(* CODESYS project mir3502tester_20200314.1.project

Project tree, tasks and I/O mapping:
  Device : Changsha Xiangji-ARM Cortex A9(xilinx zynq7000)-linux, Changsha Xiangji Hiden Technology Co.Ltd, version 3.5.10.40
    application Application
      libraries: Standard, * (System); SysFile, 3.5.15.0 (System); SysTypes2 Interfaces, * (System); SysShm, * (System); CAA Mathematics, * (CAA Technical Workgroup); CAA Net Base Services, * (CAA Technical Workgroup); SysTime, 3.5.9.0 (System); VisuDialogs, * (System); CAA Storage, 3.5.13.0 (CAA Technical Workgroup)
      task c_MainTask (cyclic, interval 20 ms, priority 20) calls prg_main
      task a_motion_tasks (cyclic, interval 10 ms, priority 5) calls EtherCAT_Master_SoftMotion.EtherCAT_Task
      program prg_main [ST]
    EtherCAT_Master_SoftMotion : EtherCAT Master SoftMotion, 3S - Smart Software Solutions GmbH, version 3.5.14.30
        settings: MasterCycleTime = 10000; MasterUseLRW = False; SlaveAutoRestart = True; NetworkName = 'eth0'; NetworkName = "eth0"; SelectNetworkByName = True; EnableTaskMessage = False; SrcAddress1 = 4784; SrcAddress2 = 3830812668
      MIR3502 : MIR3502, Cyber-MI, order no. MIR3502, version Revision=16#00000000
          settings: StationAlias = 0; DC sync0 cycletime = 10000; DC sync1 cycletime = 10000
          output Application.prg_main.mir3502_pwm01 : UINT  // PWM01-C35
          output Application.prg_main.mir3502_do00 : BIT  // DO00-C01
          input  Application.prg_main.mir3502_ai00 : UINT  // AI00-C20
          input  Application.prg_main.mir3502_di07 : BIT  // DI07-C02
          unmapped channels: PWM00-C24, DO01-C02, DO02-C03, DO03-C04, DO04-C05, DO05-C06, DO06-C07, DO07-C08, DO08-C09, DO09-C10, DO10-C11, DO11-C12, DO12-C35, DO13-C34, DO14-C33, DO15-C32, DO16-C31, DO17-C30, DO18-C29, DO19-C28, DO20-C27, DO21-C26, DO22-C25, DO23-C24, AI01-C19, AI02-C18, AI03-C17, AI04-C16, AI05-C15, AI06-C01, AI07-C02, AI08-C03, AI09-C04, AI10-C05, AI11-C06, AI12-C07, AI13-C08, AI14-C09, AI15-C10, AI16-C11,
            AI17-C12, AI18-C35, AI19-C34, AI20-C33, AI21-C32, AI22-C31, AI23-C30, AI24-C29, AI25-C28, AI26-C27, AI27-C26, AI28-C25, AI29-C24, AI30-iPWM0, AI31-iPWM1, DI00-C20, DI01-C19, DI02-C18, DI03-C17, DI04-C16, DI05-C15, DI06-C01, DI08-C03, DI09-C04, DI10-C05, DI11-C06, DI12-C07, DI13-C08, DI14-C09, DI15-C10, DI16-C11, DI17-C12, DI18-C35, DI19-C34, DI20-C33, DI21-C32, DI22-C31, DI23-C30, DI24-C29, DI25-C28,
            DI26-C27, DI27-C26, DI28-C25, DI29-C24, DI30, DI31
    IoDrvMIC7001 : IoDrvMIC7001, Cyber-MI, version 19.1.1
        unmapped channels: Ai00@C16, Ai01@C28, Ai02@C17, Ai03@C29, Ai04@C30, Ai05@C19, Ai06@C31, Ai07@C20, Ai08@C18, Ai09@D18, Ai10@D20, Ai11@D31, Ai12@D19, Ai13@D30, Ai14@D29, Ai15@D17, Ai16@D28, Ai17@D16, Ai18-Do00@C25, Ai19-Do01@C24, Ai20-Do02@C13, Ai21-Do03@C01, Ai22-Do04@C03, Ai23-Do05@C04, Ai24-Do06@C05, Ai25-Do07@C06, Ai26-Do08@C08, Ai27-Do09@C09, Ai28-Do10@C10, Ai29-Do11@C11, Ai30-Do12@D34, Ai31-Do13@D35, Ai32-Do14@D23, Ai33-Do15@D12, Ai34-Do16@D10, Ai35-Do17@D09, Ai36-Do18@D08, Ai37-Do19@D07, Ai38-Do20@D05, Ai39-Do21@D04,
          Ai40-Do22@D03, Ai41-Do23@D02, Ai42-Do24@C23, Ai43-Do25@C35, Ai44-Do26@D24, Ai45-Do27@D13, Ai46-Ao00@C22, Ai47-Ao01@D14, Ai48_Pi02, Ai49_Out5V, Ai50_VCC, Ai51_VCC_L, Ai52_VCC_R, Ai53_Pwm-i0, Ai54_Pwm-i1, Ai55_Pwm-i2, Ai56_Pwm-i3, Ai57_CPU-T, Ai58_G-x, Ai59_G-y, Ai60_G-z, Ai61-reserved, Ai62-IO-cntr, Ai63-CDS-cntr, Di00-Ai00@C16, Di01-Ai01@C28, Di02-Ai02@C17, Di03-Ai03@C29, Di04-Ai04@C30, Di05-Ai05@C19, Di06-Ai06@C31, Di07-Ai07@C20, Di08-Ai08@C18, Di09-Ai09@D18, Di10-Ai10@D20, Di11-Ai11@D31, Di12-Ai12@D19, Di13-Ai13@D30, Di14-Ai14@D29, Di15-Ai15@D17,
          Di16-Ai16@D28, Di17-Ai17@D16, Di18-Ai18@C25, Di19-Ai19@C24, Di20-Ai20@C13, Di21-Ai21@C01, Di22-Ai22@C03, Di23-Ai23@C04, Di24-Ai24@C05, Di25-Ai25@C06, Di26-Ai26@C08, Di27-Ai27@C09, Di28-Ai28@C10, Di29-Ai29@C11, Di30-Ai30@D34, Di31-Ai31@D35, Di32-Ai32@D23, Di33-Ai33@D12, Di34-Ai34@D10, Di35-Ai35@D09, Di36-Ai36@D08, Di37-Ai37@D07, Di38-Ai38@D05, Di39-Ai39@D04, Di40-Ai40@D03, Di41-Ai41@D02, Di42-Ai42@C23, Di43-Ai43@C35, Di44-Ai44@D24, Di45-Ai45@D13, Di46-Ai46@C22, Di47-Ai47@D14, Di48-Pi00@C15, Di49-Pi01@C14, Di50-Pi02@D22, Di51-Pi03@D21, Di52-reserved, Di53-reserved, Di54-reserved, Di55-reserved,
          Di56-reserved, Di57-reserved, Di58-reserved, Di59-reserved, Di60-reserved, Di61-reserved, Di62-reserved, Di63-reserved, Pi00-Di48@C15, Pi01-Di49@C14, Pi02-Di50@D22, Pi03-Di51@D21, Do00-Ai18@C25, Do01-Ai19@C24, Do02-Ai20@C13, Do03-Ai21@C01, Do04-Ai22@C03, Do05-Ai23@C04, Do06-Ai24@C05, Do07-Ai25@C06, Do08-Ai26@C08, Do09-Ai27@C09, Do10-Ai28@C10, Do11-Ai29@C11, Do12-Ai30@D34, Do13-Ai31@D35, Do14-Ai32@D23, Do15-Ai33@D12, Do16-Ai34@D10, Do17-Ai35@D09, Do18-Ai36@D08, Do19-Ai37@D07, Do20-Ai38@D05, Do21-Ai39@D04, Do22-Ai40@D03, Do23-Ai41@D02, Do24-Ai42@C23, Do25-Ai43@C35, Do26-Ai44@D24, Do27-Ai45@D13,
          Do28-Pwmi00@C33, Do29-Pwmi01@C34, Do30-Pwmi02@D25, Do31-Pwmi03@D26, PWM00@C25, PWM01@C24, PWM02@C13, PWM03@C01, PWM04@C03, PWM05@C04, PWM06@C05, PWM07@C06, PWM08@C08, PWM09@C09, PWM10@C10, PWM11@C11, PWM12@D34, PWM13@D35, PWM14@D23, PWM15@D12, PWM16@D10, PWM17@D09, PWM18@D08, PWM19@D07, PWM20@D05, PWM21@D04, PWM22@D03, PWM23@D02, PWM24@C23, PWM25@C35, PWM26@D24, PWM27@D13, PWM28-Pwmi00@C33, PWM29-Pwmi01@C34, PWM30-Pwmi02@D25, PWM31-Pwmi03@D26, PWM_I_0@C33, PWM_I_1@C34, PWM_I_2@D25, PWM_I_3@D26,
          Ao00-Ai46@C22, Ao01-Ai47@D14, LED_run, LED_err, LED_usr, ctrl_ai_raw, ctrl_adjust, ctrl_adj0, ctrl_adj1, ctrl_adj2, ctrl_adj3, ctrl_adj4
    SoftMotion General Axis Pool
      axis_4 : SM_Drive_Virtual, 3S - Smart Software Solutions GmbH, order no. 1805, version 4.0.0.0
          settings: wDriveID = 3; fSWLimitNegative = -1000.0
      axis_3 : SM_Drive_Virtual, 3S - Smart Software Solutions GmbH, order no. 1805, version 4.0.0.0
          settings: wDriveID = 2; fSWLimitNegative = -1000.0
      axis_1 : SM_Drive_Virtual, 3S - Smart Software Solutions GmbH, order no. 1805, version 4.0.0.0
          settings: wDriveID = 4
      axis_2 : SM_Drive_Virtual, 3S - Smart Software Solutions GmbH, order no. 1805, version 4.0.0.0
          settings: wDriveID = 5
  libraries: VisuSymbols, 3.5.10.0 (System)
  5ce3da45-db07-42e7-a21c-a00fff4ed8f6|C:\Users\zhou\p01.bmp
  5ce3da45-db07-42e7-a21c-a00fff4ed8f6|C:\working\p01.bmp
  5ce3da45-db07-42e7-a21c-a00fff4ed8f6|台达驱动器.jpg
  5ce3da45-db07-42e7-a21c-a00fff4ed8f6|C:\working\file.bmp
  text list GlobalTextList
  5ce3da45-db07-42e7-a21c-a00fff4ed8f6|mir3501.jpg
  text list System
  5ce3da45-db07-42e7-a21c-a00fff4ed8f6|delta.jpg
*)

// Device/Application/prg_main
PROGRAM prg_main
VAR
	mir3502_ai00:UINT;
	mir3502_pwm01:UINT;
	mir3502_di07:BOOL;
	mir3502_do00:BOOL;
	
	mydi:BOOL;
	myai:UINT;
	
	ton_io:ton;
END_VAR


ton_io(in := NOT ton_io.Q, pt := T#1S);
IF ton_io.Q THEN
	mir3502_do00 := NOT mir3502_do00;
END_IF


mir3502_pwm01 := 2048;

mydi := mir3502_di07;

myai := mir3502_ai00;

END_PROGRAM

(* text list System (id | default)
  Apr | Apr
  April | April
  Aug | Aug
  August | August
  Dec | Dec
  December | December
  Feb | Feb
  February | February
  Fri | Fri
  Friday | Friday
  Jan | Jan
  January | January
  Jul | Jul
  July | July
  Jun | Jun
  June | June
  Mar | Mar
  March | March
  May | May
  May_3Letter | May
  Mon | Mon
  Monday | Monday
  Nov | Nov
  November | November
  Oct | Oct
  October | October
  Sat | Sat
  Saturday | Saturday
  Sep | Sep
  September | September
  Sun | Sun
  Sunday | Sunday
  Thu | Thu
  Thursday | Thursday
  Tue | Tue
  Tuesday | Tuesday
  Wed | Wed
  Wednesday | Wednesday
   |  *)
